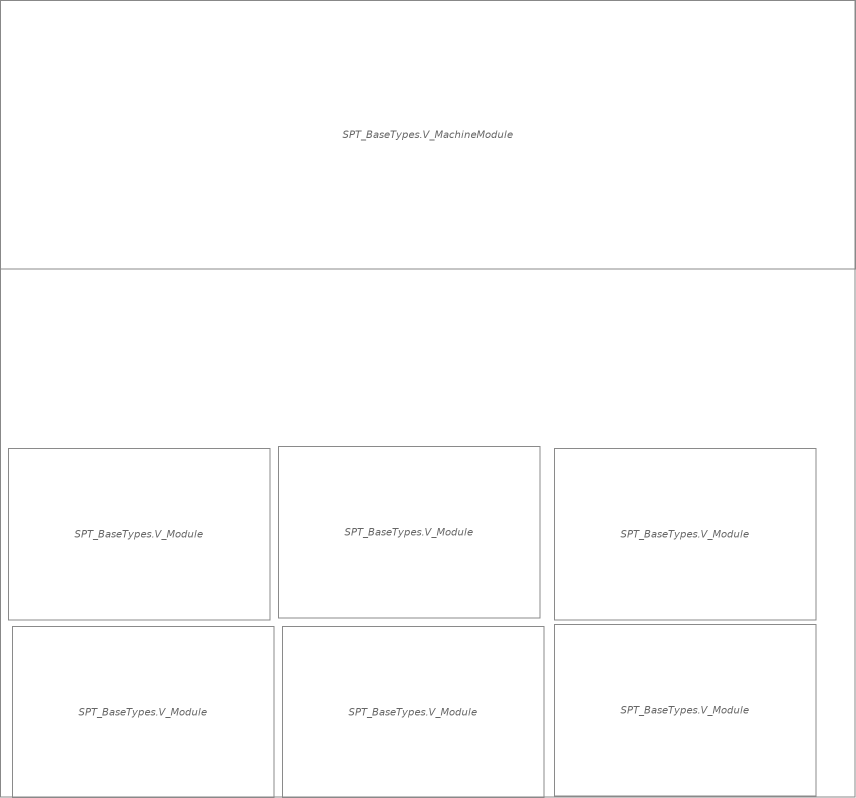
VISUALIZATION V_Machine  // 856x798
    Frame (0,0 856x269)
        shows SPT_BaseTypes.V_MachineModule(HMI := MAIN.Machine.PackMLBaseModule_HMI)
    Frame (8,448 262x172)
        shows SPT_BaseTypes.V_Module(HMI := MAIN.Machine.MainDrive.PackMLBaseModule_HMI)
    Frame (278,446 262x172)
        shows SPT_BaseTypes.V_Module(HMI := MAIN.Machine.Station1.PackMLBaseModule_HMI)
    Frame (12,626 262x172)
        shows SPT_BaseTypes.V_Module(HMI := MAIN.Machine.Station3.PackMLBaseModule_HMI)
    Frame (282,626 262x172)
        shows SPT_BaseTypes.V_Module(HMI := MAIN.Machine.Station4.PackMLBaseModule_HMI)
    Frame (554,448 262x172)
        shows SPT_BaseTypes.V_Module(HMI := MAIN.Machine.Station2.PackMLBaseModule_HMI)
    Frame (554,624 262x172)
        shows SPT_BaseTypes.V_Module(HMI := MAIN.Machine.Station5.PackMLBaseModule_HMI)
END_VISUALIZATION

(* stored: Version 1.1.0.1, ProductVersion 3.1.4024.12
   Visu V_Machine: Id {42eb1b0f-01aa-4129-b654-75b78f9759c1} *)
